// TIA Portal V19 export
DATA_BLOCK "Pu_CL01.GP08"   // DB1008
// stored: AutoNumber false, InstanceOfName Pu_Entl.GP0x, InstanceOfType FB
"Pu_Entl.GP0x"
   // VAR RETAIN
   //    In { ExternalAccessible := 'False'; ExternalVisible := 'False'; ExternalWritable := 'False'} : Struct
   //       Auto : Bool;
   //       Ein : Bool;
   //       Leckage_ok : Bool;
   //       Frg_Niv_CM05 : Bool;
   //       Betriebsart : USInt;
   //    END_STRUCT;
   //    Param { ExternalAccessible := 'False'; ExternalVisible := 'False'; ExternalWritable := 'False'} : Struct
   //       Spülzeit : Time;
   //    END_STRUCT;
   //    Zst { ExternalAccessible := 'False'; ExternalVisible := 'False'; ExternalWritable := 'False'} : Struct
   //       Niveau : USInt;
   //       Status_GP0x : USInt;
   //       Restzeit_Spülen : Time;
   //       TON_Spülventil_auf : Bool;
   //       Spuelen : Bool;
   //       Abpumpen : Bool;
   //       Bedienung_Erlaubt : Bool;
   //    END_STRUCT;
   //    Mld { ExternalAccessible := 'False'; ExternalVisible := 'False'; ExternalWritable := 'False'} : Struct
   //       Leckage : Bool;
   //       Niv_Sensorfehler : Bool;
   //       n_Auto : Bool;
   //    END_STRUCT;
   //    Out { ExternalAccessible := 'False'; ExternalVisible := 'False'; ExternalWritable := 'False'} : Struct
   //       GP0x_Ein : Bool;
   //       Spülventil : Bool;
   //    END_STRUCT;
   // END_VAR
   // VAR
   //    IEC_Timer { ExternalAccessible := 'False'; ExternalVisible := 'False'; ExternalWritable := 'False'} : Struct
   //       Leckage_ok { S7_SetPoint := 'True'} : TON_TIME;
   //       Spülventil_auf { S7_SetPoint := 'True'} : TON_TIME;
   //       Spülen { S7_SetPoint := 'True'} : TP_TIME;
   //       Leckage_niO { S7_SetPoint := 'True'} : TON_TIME;
   //    END_STRUCT;
   //    R_TRIG_Hand_EIN { ExternalAccessible := 'False'; ExternalVisible := 'False'; ExternalWritable := 'False'} : R_TRIG;
   // END_VAR
BEGIN
END_DATA_BLOCK
